{attribute 'OPC.UA.DA.StructuredType' := '1'}
TYPE ST_PumpGrundfosMagna3State :
STRUCT
	bRemoteControlOn : BOOL; //0 = control by pump, 1 = control by bus 	
	bError : BOOL; //true if pump shows an error
	bWarning : BOOL; //true if pump shows a warning
	sErrorMessage : STRING; //error code
	sWarningMessage : STRING; //warning code
	fVolumeFlowRate : REAL; //m^3/h volume flow rate from pump or external sensor
	fTemperatureInternal : REAL; //°C
	fTemperatureExternal : REAL; //°C
	fTemperatureDifference : REAL; //°C
	fPressureDifference : REAL; //pa = 10^-5 bar
	fPowerElectric : REAL; //W
	fPowerHydraulic : REAL; //W
	fPowerThermal : REAL; //W
	fRotationalSpeed : REAL; //rpm
END_STRUCT
END_TYPE

(* stored: Version 1.1.0.1, ProductVersion 3.1.4024.10
   DUT ST_PumpGrundfosMagna3State: Id {2e0e0d05-2e8a-40b3-8fdf-0cb5e297c45b} *)
